// TIA Portal V17 export
// export: Created 2025-03-05T08:01:03.4001767Z, ExportSetting WithDefaults, DisplayName Totally Integrated Automation Portal, DisplayVersion V17 Update 8, DisplayName TIA Portal Openness, DisplayVersion V17 Update 8, DisplayName TIA Portal Version Control Interface, DisplayVersion V17, DisplayName SINAMICS Startdrive Advanced, DisplayVersion V17 SP2, DisplayName SINAMICS Startdrive G110M, G120, G120C, G120D, G120P, G115D, DisplayVersion V17 SP2, DisplayName SINAMICS Startdrive G130, G150, S120, S150, SINAMICS MV, S210, DisplayVersion V17 SP2, DisplayName STEP 7 Professional, DisplayVersion V17 Update 8, DisplayName SINUMERIK ONE STEP 7 Toolbox, DisplayVersion V17 Update 12, DisplayName SINUMERIK 840D sl STEP 7 Toolbox, DisplayVersion V17 Update 12, DisplayName STEP 7 Safety, DisplayVersion V17 Update 6, DisplayName WinCC Advanced, DisplayVersion V17 Update 8
FUNCTION_BLOCK "FB1016_SAFETY_DOORS"   // FB1016, F_LAD
{ S7_Optimized_Access := 'TRUE' }
AUTHOR : ETXETAR
VERSION : 1.0
// stored: AutoNumber false, IsIECCheckEnabled false, UDAEnableTagReadback false
   VAR_INPUT
      FEEDBACK_OFF_SAFETY_DOORS_IN : Bool;   // FEEDBACK OFF SAFETY DOORS
      FEEDBACK_OFF_E_SAFE_DOORS_RST_STR_IN : Bool;   // FEEDBACK OFF SAFETY DOORS RESET START INPUT
      DOOR_1 : Bool;   // DOOR 1 INPUT
      DOOR_2 : Bool;   // DOOR 2 INPUT
      DOOR_3 : Bool;   // DOOR 3 INPUT
      DOOR_4 : Bool;   // DOOR 4 INPUT
      DOOR_5 : Bool;   // DOOR 5 INPUT
      DOOR_6 : Bool;   // DOOR 6 INPUT
      DOOR_7 : Bool;   // DOOR 7 INPUT
      DOOR_8 : Bool;   // DOOR 8 INPUT
      DOOR_9 : Bool;   // DOOR 9 INPUT
      DOOR_10 : Bool;   // DOOR 10 INPUT
   END_VAR
   VAR_OUTPUT
      SAFE_DOORS_CLOSED_LOCKED : Bool;   // SAFETY DOORS CLOSED AND LOCKED OUTPUT
      SAFE_DOORS_CLOSED_LOCKED_DEL2 : Bool;   // SAFETY DOORS CLOSED AND LOCKED DELAYED 2 OUTPUT
      SAFE_DOORS_CLOSED_LOCKED_DEL3 : Bool;   // SAFETY DOORS CLOSED AND LOCKED DELAYED 3 OUTPUT
      SAFE_DOORS_CLOSED_LOCKED_DEL4 : Bool;   // SAFETY DOORS CLOSED AND LOCKED DELAYED 4 OUTPUT
      FEEDBACK_ERROR : Bool;   // SAFETY DOORS CLOSED AND LOCKED FEEDBACK ERROR
   END_VAR
   VAR
      ALL_DOORS_CLOSED_AND_LOCKED : Bool;   // ALL DOORS CLOSED AND LOCKED
      SAFE_GATES_CLOSED_AND_LOCKED_RESET : Bool;   // MACHINE SAFETY GATES CLOSED AND LOCKED RESET
      SAFE_GATES_CLOSED_AND_LOCKED_RESET_REQ : Bool;   // MACHINE SAFETY GATES CLOSED AND LOCKED RESET REQUEST
      FEEDBACK_OFF_OK : Bool;   // SAFETY DOORS FEEDBACK OFF OK
      SFDOOR_Instance : SFDOOR;
      F_DOOR_DEL2_Timer_Instance : TOF;
      F_DOOR_DEL3_Timer_Instance : TOF;
      F_DOOR_DEL4_Timer_Instance : TOF;
      FDBACK_Instance : FDBACK;
      F_IEC_Timer_FEEDBACK : TON;
   END_VAR
   // F_IEC_Timer_FEEDBACK.PT := T#30ms;
BEGIN

REGION Network 1: ALL DOORS CLOSED AND LOCKED
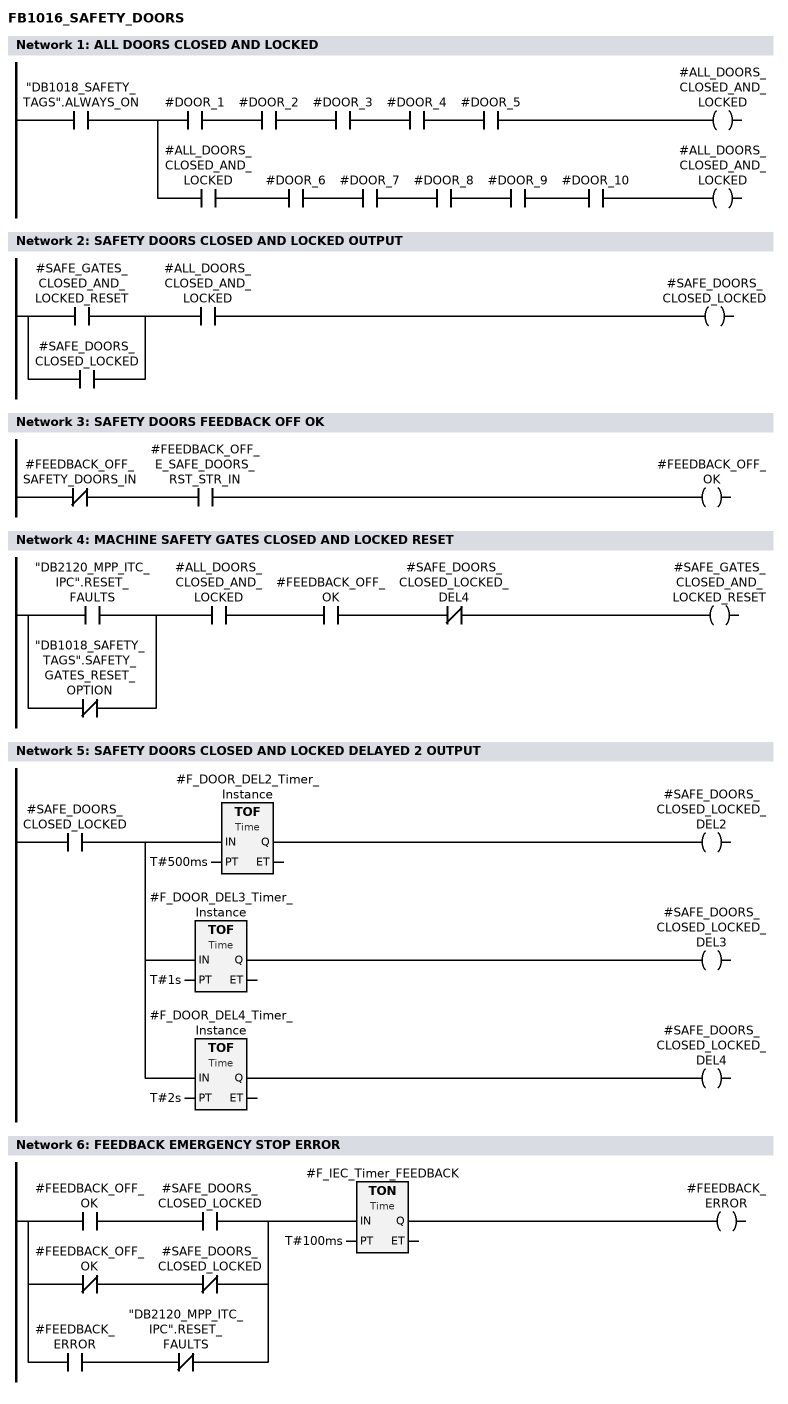
   RUNG wire#powerrail
      Contact( "DB1018_SAFETY_TAGS".ALWAYS_ON )
      wire#w1
      Contact( #DOOR_1 )
      Contact( #DOOR_2 )
      Contact( #DOOR_3 )
      Contact( #DOOR_4 )
      Contact( #DOOR_5 )
      Coil( #ALL_DOORS_CLOSED_AND_LOCKED )
   END_RUNG
   RUNG wire#w1
      Contact( #ALL_DOORS_CLOSED_AND_LOCKED )
      Contact( #DOOR_6 )
      Contact( #DOOR_7 )
      Contact( #DOOR_8 )
      Contact( #DOOR_9 )
      Contact( #DOOR_10 )
      Coil( #ALL_DOORS_CLOSED_AND_LOCKED )
   END_RUNG
   // the same network as SCL:
   #ALL_DOORS_CLOSED_AND_LOCKED := "DB1018_SAFETY_TAGS".ALWAYS_ON AND #DOOR_1 AND #DOOR_2 AND #DOOR_3 AND #DOOR_4 AND #DOOR_5;
   #ALL_DOORS_CLOSED_AND_LOCKED := "DB1018_SAFETY_TAGS".ALWAYS_ON AND #ALL_DOORS_CLOSED_AND_LOCKED AND #DOOR_6 AND #DOOR_7 AND #DOOR_8 AND #DOOR_9 AND #DOOR_10;
END_REGION

REGION Network 2: SAFETY DOORS CLOSED AND LOCKED OUTPUT
   RUNG wire#powerrail
      Contact( #SAFE_GATES_CLOSED_AND_LOCKED_RESET )
      wire#w1
      Contact( #ALL_DOORS_CLOSED_AND_LOCKED )
      Coil( #SAFE_DOORS_CLOSED_LOCKED )
   END_RUNG
   RUNG wire#powerrail
      Contact( #SAFE_DOORS_CLOSED_LOCKED )
   END_RUNG wire#w1
   // the same network as SCL:
   #SAFE_DOORS_CLOSED_LOCKED := (#SAFE_GATES_CLOSED_AND_LOCKED_RESET OR #SAFE_DOORS_CLOSED_LOCKED) AND #ALL_DOORS_CLOSED_AND_LOCKED;
END_REGION

REGION Network 3: SAFETY DOORS FEEDBACK OFF OK
   RUNG wire#powerrail
      I_Contact( #FEEDBACK_OFF_SAFETY_DOORS_IN )
      Contact( #FEEDBACK_OFF_E_SAFE_DOORS_RST_STR_IN )
      Coil( #FEEDBACK_OFF_OK )
   END_RUNG
   // the same network as SCL:
   #FEEDBACK_OFF_OK := NOT #FEEDBACK_OFF_SAFETY_DOORS_IN AND #FEEDBACK_OFF_E_SAFE_DOORS_RST_STR_IN;
END_REGION

REGION Network 4: MACHINE SAFETY GATES CLOSED AND LOCKED RESET
   RUNG wire#powerrail
      Contact( "DB2120_MPP_ITC_IPC".RESET_FAULTS )
      wire#w1
      Contact( #ALL_DOORS_CLOSED_AND_LOCKED )
      Contact( #FEEDBACK_OFF_OK )
      I_Contact( #SAFE_DOORS_CLOSED_LOCKED_DEL4 )
      Coil( #SAFE_GATES_CLOSED_AND_LOCKED_RESET )
   END_RUNG
   RUNG wire#powerrail
      I_Contact( "DB1018_SAFETY_TAGS".SAFETY_GATES_RESET_OPTION )
   END_RUNG wire#w1
   // the same network as SCL:
   #SAFE_GATES_CLOSED_AND_LOCKED_RESET := ("DB2120_MPP_ITC_IPC".RESET_FAULTS OR NOT "DB1018_SAFETY_TAGS".SAFETY_GATES_RESET_OPTION) AND #ALL_DOORS_CLOSED_AND_LOCKED AND #FEEDBACK_OFF_OK AND NOT #SAFE_DOORS_CLOSED_LOCKED_DEL4;
END_REGION

REGION Network 5: SAFETY DOORS CLOSED AND LOCKED DELAYED 2 OUTPUT
   RUNG wire#powerrail
      Contact( #SAFE_DOORS_CLOSED_LOCKED )
      wire#w1
      { S7_Templates := "[time_type := Time, codedbool_type := DInt]" } #F_DOOR_DEL2_Timer_Instance.TOF(pt := T#500ms, et =>)
      Coil( #SAFE_DOORS_CLOSED_LOCKED_DEL2 )
   END_RUNG
   RUNG wire#w1
      { S7_Templates := "[time_type := Time, codedbool_type := DInt]" } #F_DOOR_DEL3_Timer_Instance.TOF(pt := T#1s, et =>)
      Coil( #SAFE_DOORS_CLOSED_LOCKED_DEL3 )
   END_RUNG
   RUNG wire#w1
      { S7_Templates := "[time_type := Time, codedbool_type := DInt]" } #F_DOOR_DEL4_Timer_Instance.TOF(pt := T#2s, et =>)
      Coil( #SAFE_DOORS_CLOSED_LOCKED_DEL4 )
   END_RUNG
   // the same network as SCL:
   #F_DOOR_DEL2_Timer_Instance.TOF(IN := #SAFE_DOORS_CLOSED_LOCKED, PT := T#500ms);
   #SAFE_DOORS_CLOSED_LOCKED_DEL2 := #F_DOOR_DEL2_Timer_Instance.Q;
   #F_DOOR_DEL3_Timer_Instance.TOF(IN := #SAFE_DOORS_CLOSED_LOCKED, PT := T#1s);
   #SAFE_DOORS_CLOSED_LOCKED_DEL3 := #F_DOOR_DEL3_Timer_Instance.Q;
   #F_DOOR_DEL4_Timer_Instance.TOF(IN := #SAFE_DOORS_CLOSED_LOCKED, PT := T#2s);
   #SAFE_DOORS_CLOSED_LOCKED_DEL4 := #F_DOOR_DEL4_Timer_Instance.Q;
END_REGION

REGION Network 6: FEEDBACK EMERGENCY STOP ERROR
   RUNG wire#powerrail
      Contact( #FEEDBACK_OFF_OK )
      Contact( #SAFE_DOORS_CLOSED_LOCKED )
      wire#w1
      { S7_Templates := "[time_type := Time, codedbool_type := DInt]" } #F_IEC_Timer_FEEDBACK.TON(pt := T#100ms, et =>)
      Coil( #FEEDBACK_ERROR )
   END_RUNG
   RUNG wire#powerrail
      I_Contact( #FEEDBACK_OFF_OK )
      I_Contact( #SAFE_DOORS_CLOSED_LOCKED )
   END_RUNG wire#w1
   RUNG wire#powerrail
      Contact( #FEEDBACK_ERROR )
      I_Contact( "DB2120_MPP_ITC_IPC".RESET_FAULTS )
   END_RUNG wire#w1
   // the same network as SCL:
   #F_IEC_Timer_FEEDBACK.TON(IN := (#FEEDBACK_OFF_OK AND #SAFE_DOORS_CLOSED_LOCKED) OR (NOT #FEEDBACK_OFF_OK AND NOT #SAFE_DOORS_CLOSED_LOCKED) OR (#FEEDBACK_ERROR AND NOT "DB2120_MPP_ITC_IPC".RESET_FAULTS),
                           PT := T#100ms);
   #FEEDBACK_ERROR := #F_IEC_Timer_FEEDBACK.Q;
END_REGION
END_FUNCTION_BLOCK
